{attribute 'reflection'} 
FUNCTION_BLOCK PUBLIC T_InstanceNameBase
VAR
  {attribute 'instance-path'} 
  {attribute 'noinit'} 
  name : T_MaxString;
  
  _instanceName : T_MaxString;
  isInstanceNameSet : BOOL := FALSE;
END_VAR

PROPERTY FINAL InstanceName : T_MaxString; // returns the fully scoped variable name
GET
IF NOT isInstanceNameSet THEN
   setInstanceName();
END_IF

InstanceName := _instanceName;
END_GET
END_PROPERTY

METHOD PRIVATE SetInstanceName
VAR
	charsToDeleteFromPath : INT;
END_VAR
//Remove Solution_Name
charsToDeleteFromPath := FIND(name, '.');
_instanceName := DELETE(name, charsToDeleteFromPath, 1);
//Remove ProjectName
charsToDeleteFromPath := FIND(_instanceName, '.');
//gives us just "FirstDeclaredPOU.etc.etc..." from above.
_instanceName := DELETE(_instanceName, charsToDeleteFromPath, 1);
END_METHOD

END_FUNCTION_BLOCK

(* stored: Version 1.1.0.1, ProductVersion 3.1.4024.12
   POU T_InstanceNameBase: Id {b74b87ab-3edd-0d49-06ea-12f9876971cc}, SpecialFunc None
   Property InstanceName: Id {1ec45583-ccb3-01f2-0d0a-04356f36a10b}
   Get Get: Id {0e8c4cf6-5109-0537-1e3d-136fdc1f01c0}
   Method SetInstanceName: Id {fe0a3aab-cec0-0aee-38ee-b90839220926} *)
